# EPICS autosave request: iocBoot/iocLinux/auto_settings.req
file "mca_settings.req",      P=$(P), M=aim_adc1
file "mca_settings.req",      P=$(P), M=aim_adc2
file "icb_amp_settings.req",  P=$(P), AMP=amp1
file "icb_adc_settings.req",  P=$(P), ADC=adc1
#file "icb_hvps_settings.req", P=$(P), HVPS=hvps1
file "icb_tca_settings.req",  P=$(P), TCA=tca1
